(* PLC project SafeLOGIC-1, BrAutomation SafeDESIGNER  4.4.0.0 *)
(* stored: companyURL http://www.br-automation.com, creationDateTime Thu Mar 18 12:04:02 2021 *)

PROGRAM Main
  VAR  (* added by the conversion: wires and edge detectors of the diagram *)
    _SAFEBOOL_TO_BOOL24_OUT : BOOL;
  END_VAR

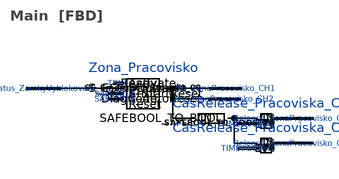
(* FBD diagram, written out as Structured Text *)
Zona_Pracovisko(Activate := TRUE, S_EStopIn := Status_ZamkyVyblokovane, S_StartReset := SAFETRUE, S_AutoReset := SAFETRUE);
SO_ZonaPracovisko_CH2 := Zona_Pracovisko.S_EStopOut;
SO_ZonaPracovisko_CH1 := Zona_Pracovisko.S_EStopOut;
_SAFEBOOL_TO_BOOL24_OUT := SAFEBOOL_TO_BOOL(Zona_Pracovisko.S_EStopOut);
CasRelease_Pracoviska_CH1(IN := _SAFEBOOL_TO_BOOL24_OUT, PT := TIME#500ms);
Release_ZonaPracovisko_CH1 := CasRelease_Pracoviska_CH1.Q;
CasRelease_Pracoviska_CH2(IN := _SAFEBOOL_TO_BOOL24_OUT, PT := TIME#500ms);
Release_ZonaPracovisko_CH2 := CasRelease_Pracoviska_CH2.Q;
END_PROGRAM
